// TIA Portal V17 export
// export: Created 2024-08-26T21:10:53.653086Z, ExportSetting WithDefaults, DisplayName Totally Integrated Automation Portal, DisplayVersion V17 Update 7, DisplayName TIA Portal Openness, DisplayVersion V17 Update 7, DisplayName TIA Portal Version Control Interface, DisplayVersion V17, DisplayName SINAMICS Startdrive Advanced, DisplayVersion V17 SP2, DisplayName SINAMICS Startdrive G110M, G120, G120C, G120D, G120P, G115D, DisplayVersion V17 SP2, DisplayName SINAMICS Startdrive G130, G150, S120, S150, SINAMICS MV, S210, DisplayVersion V17 SP2, DisplayName STEP 7 Professional, DisplayVersion V17 Update 7, DisplayName STEP 7 Safety, DisplayVersion V17 Update 6, DisplayName WinCC Advanced / Unified PC, DisplayVersion V17 Update 7
VAR_GLOBAL   // PLC tag table "digitalFieldbusOutputs"
   qcylinder1DirectionA AT %Q149.0 : Bool;
   qcylinder1DirectionB AT %Q151.0 : Bool;
   qcylinder2DirectionA AT %Q149.1 : Bool;
   qcylinder2DirectionB AT %Q151.1 : Bool;
   qcylinder7DirectionA AT %Q701.2 : Bool;
   qcylinder7DirectionB AT %Q701.3 : Bool;
   qcylinder4DirectionA AT %Q149.3 : Bool;
   qcylinder4DirectionB AT %Q151.3 : Bool;
   qcylinder5DirectionA AT %Q149.4 : Bool;
   qcylinder5DirectionB AT %Q151.4 : Bool;
   qcylinder6DirectionA AT %Q149.5 : Bool;
   qcylinder6DirectionB AT %Q151.5 : Bool;
   qcylinder3DirectionA AT %Q149.2 : Bool;
   qcylinder3DirectionB AT %Q151.2 : Bool;
   qcylinder8DirectionA AT %Q701.4 : Bool;
   qcylinder8DirectionB AT %Q701.5 : Bool;
   qcylinder9DirectionA AT %Q701.6 : Bool;
   qcylinder9DirectionB AT %Q701.7 : Bool;
   qcylinder10DirectionA AT %Q702.0 : Bool;
   qcylinder10DirectionB AT %Q702.1 : Bool;
   qActivateCutOffValve AT %Q147.7 : Bool;
END_VAR
